PROGRAM MAIN
VAR
    bTest : BOOL;
END_VAR

END_PROGRAM

(* stored: Version 1.1.0.1, ProductVersion 3.1.4024.12
   POU MAIN: Id {500fed89-99c1-41f9-aaf6-95df3ebe7e5f}, SpecialFunc None *)
